// Mitsubishi GX Works2 project: 타이머응용1   PLC: Q02/Q02H

PROGRAM MAIN
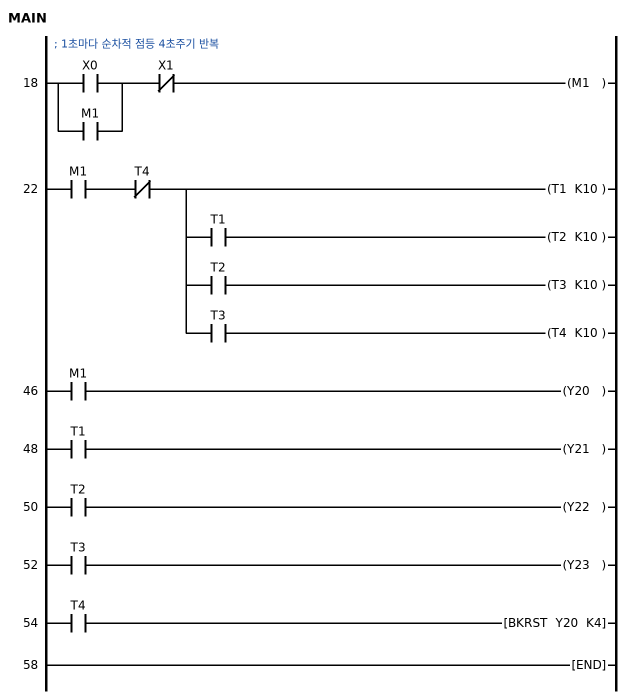
; 1초마다 순차적 점등 4초주기 반복
18    LD      X0
      OR      M1
      ANI     X1
      OUT     M1
22    LD      M1
      ANI     T4
      OUT     T1 K10
      MPS
      AND     T1
      OUT     T2 K10
      MRD
      AND     T2
      OUT     T3 K10
      MPP
      AND     T3
      OUT     T4 K10
46    LD      M1
      OUT     Y20
48    LD      T1
      OUT     Y21
50    LD      T2
      OUT     Y22
52    LD      T3
      OUT     Y23
54    LD      T4
      BKRST   Y20 K4
58    END
END_PROGRAM
